{attribute 'reflection'} 
FUNCTION_BLOCK FB_EventLogger EXTENDS TcLog
VAR
	_WorkString			: Tc2_System.T_MaxString;
	isSpammable			: BOOL;
	
	sStringToBeLogged : T_MaxString;
	OldsCompletedString, NewCompletedString : T_MaxString;
END_VAR

METHOD Append : REFERENCE TO FB_EventLogger
VAR_INPUT
	sString		: T_MaxString;
END_VAR

VAR_INST
	OldString 	: T_MaxString;
END_VAR
_WorkString := CONCAT(_WorkString, sString);

Append REF= THIS^;
END_METHOD

METHOD CanSpam : REFERENCE TO FB_EventLogger
VAR
	
END_VAR
isSpammable := TRUE; 
CanSpam REF= THIS^;
END_METHOD

/// Logs the log string in DEBUG level.
METHOD Debug : BOOL
VAR_INPUT
  	message : T_MaxString; 
END_VAR
_WorkString := CONCAT(_WorkString, message);
NewCompletedString := _WorkString;
_WorkString := '';

IF NewCompletedString <> OldsCompletedString OR isSpammable THEN
	SUPER^.Debug(NewCompletedString);
	OldsCompletedString := NewCompletedString;
	isSpammable := FALSE;
END_IF
END_METHOD

/// Logs the log string in ERROR level.
METHOD Error : BOOL
VAR_INPUT
  	message : T_MaxString; 
END_VAR
_WorkString := CONCAT(_WorkString, message);
NewCompletedString := _WorkString;
_WorkString := '';

IF NewCompletedString <> OldsCompletedString THEN
	SUPER^.Error(NewCompletedString);
	OldsCompletedString := NewCompletedString;
	isSpammable := FALSE;
END_IF
END_METHOD

/// Logs the log string in FATAL level.
METHOD Fatal : BOOL
VAR_INPUT
  	message : T_MaxString; 
END_VAR
_WorkString := CONCAT(_WorkString, message);
NewCompletedString := _WorkString;
_WorkString := '';

IF NewCompletedString <> OldsCompletedString THEN
	SUPER^.Error(NewCompletedString);
	OldsCompletedString := NewCompletedString;
	isSpammable := FALSE;
END_IF
END_METHOD

/// Logs the log string in INFORMATION level.
METHOD Information : BOOL
VAR_INPUT
  	message : T_MaxString; 
END_VAR
_WorkString := CONCAT(_WorkString, message);
NewCompletedString := _WorkString;
_WorkString := '';

IF NewCompletedString <> OldsCompletedString THEN
	SUPER^.Information(NewCompletedString);
	OldsCompletedString := NewCompletedString;
	isSpammable := FALSE;
END_IF
END_METHOD

/// Logs the log string in WARNING level.
METHOD Warning : BOOL
VAR_INPUT
  	message : T_MaxString; 
END_VAR
_WorkString := CONCAT(_WorkString, message);
NewCompletedString := _WorkString;
_WorkString := '';

IF NewCompletedString <> OldsCompletedString THEN
	SUPER^.Warning(NewCompletedString);
	OldsCompletedString := NewCompletedString;
	isSpammable := FALSE;
END_IF
END_METHOD

END_FUNCTION_BLOCK

(* stored: Version 1.1.0.1, ProductVersion 3.1.4024.12
   POU FB_EventLogger: Id {1aa67368-e303-4734-ae87-07290b7c16e8}, SpecialFunc None
   Method Append: Id {d1e5fd85-235d-459a-b497-045db3674c42}
   Method CanSpam: Id {a8d029d9-2b0c-4158-b488-9f9e8e28e4e7}
   Method Debug: Id {5999ae39-e738-46af-b0a3-2337db0b32f0}
   Method Error: Id {37e1358a-40dd-4b42-87ad-97f7d6613f51}
   Method Fatal: Id {129abf48-7d5e-4c65-98c8-de9c267bdd5c}
   Method Information: Id {6991a8ac-5536-40b5-a57a-056ccac01b8d}
   Method Warning: Id {b6254e94-446f-4182-8668-824bf93459ce} *)
